{attribute addProperty BoxType "EK1100-0000-0018"}
{attribute addProperty Id "Beckhoff_ER2xxxEK1122Beckhoff_ER2xxxEK1122_89F8FCAB7280910"}
{attribute addProperty CRC "1795394176"}
{attribute addProperty SizeInBites "7280"}
{attribute addProperty SizeInBytes "910"}
TYPE Beckhoff_ER2xxx_6B038A80 EXTENDS EK1100_179A0949 :
STRUCT
	{attribute addProperty Name "Beckhoff_ER2xxxEK1122"}
	Beckhoff_ER2xxxEK1122 : Beckhoff_ER2xxxEK1122_89F8FCAB;
END_STRUCT
END_TYPE

(* stored: Version 1.2.0.0, ProductVersion 3.1.4024.9
   DUT Beckhoff_ER2xxx_6B038A80: Id {ceb0faa9-7f8e-49ca-bbe7-f065a63a1a90} *)
